Fanuc KAREL source: kc00012.KL

-- PROVISIONAL review KL for V1013-1; original PC SHA256 785bf375a0fd5870a480d48840b6f32017e40dee7a3841cbb92b19c24914e7f5
-- Incomplete behavior may be omitted. Consult companion uncertainty JSON. Do not deploy.
PROGRAM KC00012
%NOLOCKGROUP
BEGIN
  -- UNRESOLVED_PC offsets 5-51; opcodes 27,22,22,22,22,22,22,22,31
  -- UNRESOLVED_PC offsets 56-60; opcodes 7F
END KC00012
